FUNCTION_BLOCK FB_StringLookupINTMock EXTENDS FB_FallibleMock IMPLEMENTS I_StringLookupINT
VAR
    nValue : INT;
END_VAR


METHOD Lookup : INT
VAR_INPUT
    sLookup	: STRING;
END_VAR

Lookup := nValue;
END_METHOD


METHOD SetValid

ClearError();
END_METHOD

END_FUNCTION_BLOCK

(* stored: Version 1.1.0.1
   POU FB_StringLookupINTMock: Id {d0b4a7e9-2d3c-4985-b1c8-bb2c34a08f90}, SpecialFunc None
   Method Lookup: Id {5c037a72-ea45-45f3-9d22-aab555885a73}
   Method SetValid: Id {f5e0b920-bdf0-4251-957b-b2087937d68e} *)
